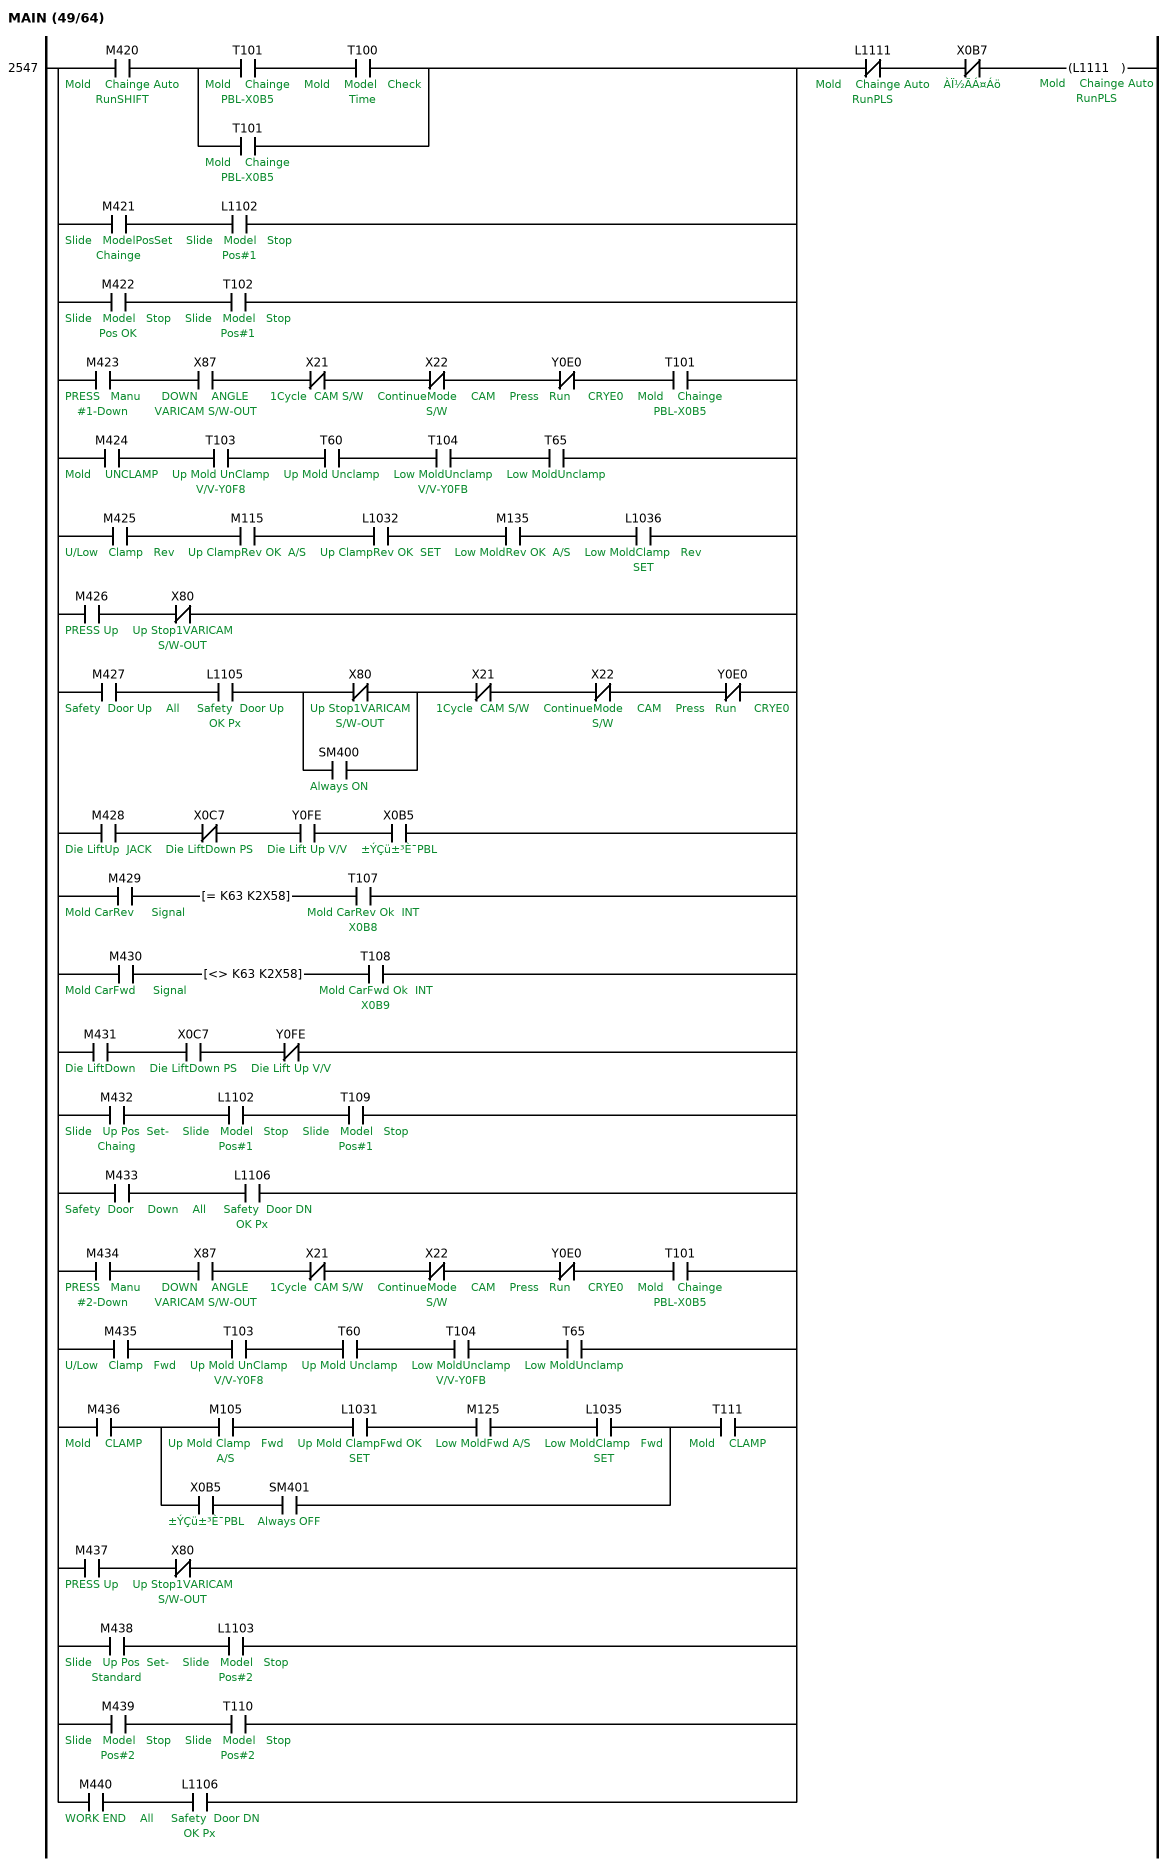
[picture p48: ladder of MAIN, rungs at steps 2547 to 2547]
2547  LD      M420  ; Mold    Chainge Auto RunSHIFT
      LD      T101  ; Mold    Chainge PBL-X0B5
      AND     T100  ; Mold    Model   Check   Time
      OR      T101  ; Mold    Chainge PBL-X0B5
      ANB
      LD      M421  ; Slide   ModelPosSet     Chainge
      AND     L1102  ; Slide   Model   Stop    Pos#1
      ORB
      LD      M422  ; Slide   Model   Stop    Pos OK
      AND     T102  ; Slide   Model   Stop    Pos#1
      ORB
      LD      M423  ; PRESS   Manu #1-Down
      AND     X87  ; DOWN    ANGLE   VARICAM S/W-OUT
      ANI     X21  ; 1Cycle  CAM S/W
      ANI     X22  ; ContinueMode    CAM S/W
      ANI     Y0E0  ; Press   Run     CRYE0
      AND     T101  ; Mold    Chainge PBL-X0B5
      ORB
      LD      M424  ; Mold    UNCLAMP
      AND     T103  ; Up Mold UnClamp V/V-Y0F8
      AND     T60  ; Up Mold Unclamp
      AND     T104  ; Low MoldUnclamp V/V-Y0FB
      AND     T65  ; Low MoldUnclamp
      ORB
      LD      M425  ; U/Low   Clamp   Rev
      AND     M115  ; Up ClampRev OK  A/S
      AND     L1032  ; Up ClampRev OK  SET
      AND     M135  ; Low MoldRev OK  A/S
      AND     L1036  ; Low MoldClamp   Rev SET
      ORB
      LD      M426  ; PRESS Up
      ANI     X80  ; Up Stop1VARICAM S/W-OUT
      ORB
      LD      M427  ; Safety  Door Up
      AND     L1105  ; All     Safety  Door Up OK Px
      LDI     X80  ; Up Stop1VARICAM S/W-OUT
      OR      SM400  ; Always ON
      ANB
      ANI     X21  ; 1Cycle  CAM S/W
      ANI     X22  ; ContinueMode    CAM S/W
      ANI     Y0E0  ; Press   Run     CRYE0
      ORB
      LD      M428  ; Die LiftUp  JACK
      ANI     X0C7  ; Die LiftDown PS
      AND     Y0FE  ; Die Lift Up V/V
      AND     X0B5  ; ±ÝÇü±³È¯PBL
      ORB
      LD      M429  ; Mold CarRev     Signal
      AND=    K63 K2X58
      AND     T107  ; Mold CarRev Ok  INT X0B8
      ORB
      LD      M430  ; Mold CarFwd     Signal
      AND<>   K63 K2X58
      AND     T108  ; Mold CarFwd Ok  INT X0B9
      ORB
      LD      M431  ; Die LiftDown
      AND     X0C7  ; Die LiftDown PS
      ANI     Y0FE  ; Die Lift Up V/V
      ORB
      LD      M432  ; Slide   Up Pos  Set-    Chaing
      AND     L1102  ; Slide   Model   Stop    Pos#1
      AND     T109  ; Slide   Model   Stop    Pos#1
      ORB
      LD      M433  ; Safety  Door    Down
      AND     L1106  ; All     Safety  Door DN OK Px
      ORB
      LD      M434  ; PRESS   Manu #2-Down
      AND     X87  ; DOWN    ANGLE   VARICAM S/W-OUT
      ANI     X21  ; 1Cycle  CAM S/W
      ANI     X22  ; ContinueMode    CAM S/W
      ANI     Y0E0  ; Press   Run     CRYE0
      AND     T101  ; Mold    Chainge PBL-X0B5
      ORB
      LD      M435  ; U/Low   Clamp   Fwd
      AND     T103  ; Up Mold UnClamp V/V-Y0F8
      AND     T60  ; Up Mold Unclamp
      AND     T104  ; Low MoldUnclamp V/V-Y0FB
      AND     T65  ; Low MoldUnclamp
      ORB
      LD      M436  ; Mold    CLAMP
      LD      M105  ; Up Mold Clamp   Fwd A/S
      AND     L1031  ; Up Mold ClampFwd OK  SET
      AND     M125  ; Low MoldFwd A/S
      AND     L1035  ; Low MoldClamp   Fwd SET
      LD      X0B5  ; ±ÝÇü±³È¯PBL
      AND     SM401  ; Always OFF
      ORB
      ANB
      AND     T111  ; Mold    CLAMP
      ORB
      LD      M437  ; PRESS Up
      ANI     X80  ; Up Stop1VARICAM S/W-OUT
      ORB
      LD      M438  ; Slide   Up Pos  Set-    Standard
      AND     L1103  ; Slide   Model   Stop    Pos#2
      ORB
      LD      M439  ; Slide   Model   Stop    Pos#2
      AND     T110  ; Slide   Model   Stop    Pos#2
      ORB
      LD      M440  ; WORK END
      AND     L1106  ; All     Safety  Door DN OK Px
      ORB
      ANI     L1111  ; Mold    Chainge Auto RunPLS
      ANI     X0B7  ; ÀÏ½ÃÁ¤Áö
      OUT     L1111  ; Mold    Chainge Auto RunPLS
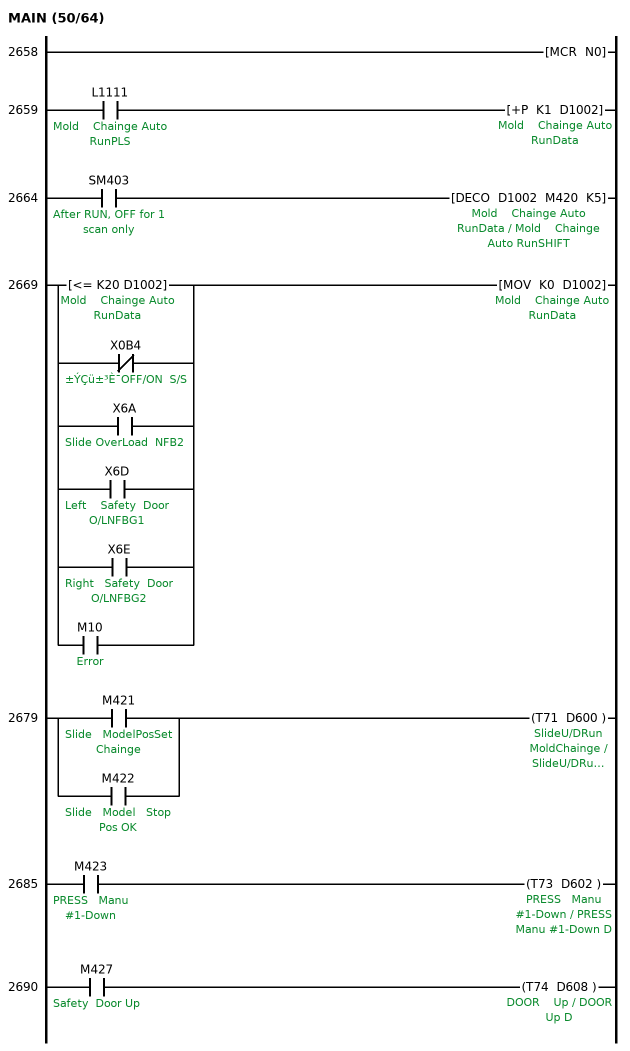
2658  MCR     N0
2659  LD      L1111  ; Mold    Chainge Auto RunPLS
      +P      K1 D1002  ; Mold    Chainge Auto RunData
2664  LD      SM403  ; After RUN, OFF for 1 scan only
      DECO    D1002 M420 K5
2669  LD<=    K20 D1002  ; Mold    Chainge Auto RunData
      ORI     X0B4  ; ±ÝÇü±³È¯OFF/ON  S/S
      OR      X6A  ; Slide OverLoad  NFB2
      OR      X6D  ; Left    Safety  Door O/LNFBG1
      OR      X6E  ; Right   Safety  Door O/LNFBG2
      OR      M10  ; Error
      MOV     K0 D1002
2679  LD      M421  ; Slide   ModelPosSet     Chainge
      OR      M422  ; Slide   Model   Stop    Pos OK
      OUT     T71 D600  ; SlideU/DRun MoldChainge / SlideU/DRun MoldChainge
2685  LD      M423  ; PRESS   Manu #1-Down
      OUT     T73 D602  ; PRESS   Manu #1-Down / PRESS   Manu #1-Down D
2690  LD      M427  ; Safety  Door Up
      OUT     T74 D608  ; DOOR    Up / DOOR    Up D
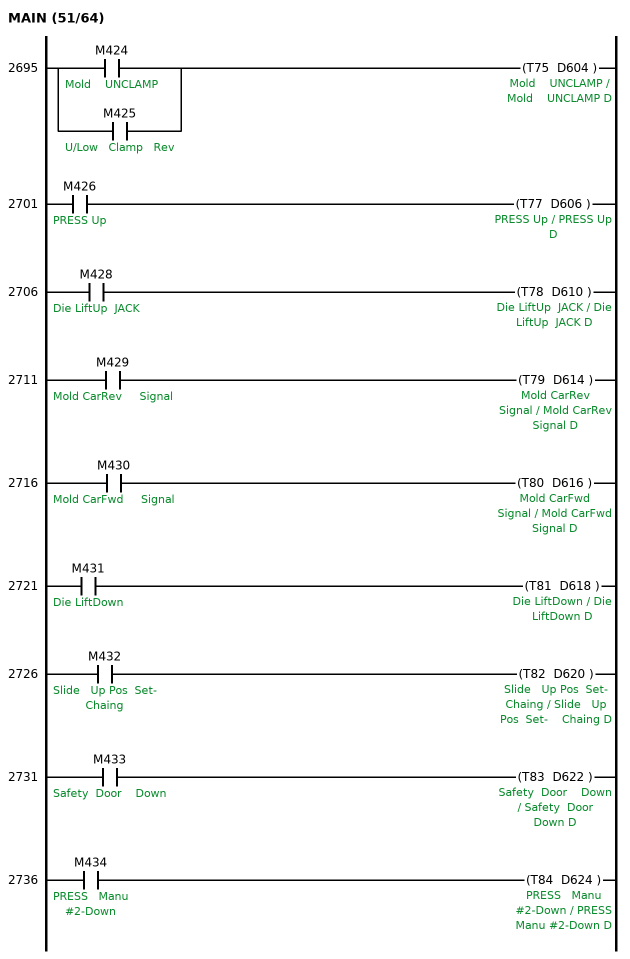
2695  LD      M424  ; Mold    UNCLAMP
      OR      M425  ; U/Low   Clamp   Rev
      OUT     T75 D604  ; Mold    UNCLAMP / Mold    UNCLAMP D
2701  LD      M426  ; PRESS Up
      OUT     T77 D606  ; PRESS Up / PRESS Up D
2706  LD      M428  ; Die LiftUp  JACK
      OUT     T78 D610  ; Die LiftUp  JACK / Die LiftUp  JACK D
2711  LD      M429  ; Mold CarRev     Signal
      OUT     T79 D614  ; Mold CarRev     Signal / Mold CarRev     Signal D
2716  LD      M430  ; Mold CarFwd     Signal
      OUT     T80 D616  ; Mold CarFwd     Signal / Mold CarFwd     Signal D
2721  LD      M431  ; Die LiftDown
      OUT     T81 D618  ; Die LiftDown / Die LiftDown D
2726  LD      M432  ; Slide   Up Pos  Set-    Chaing
      OUT     T82 D620  ; Slide   Up Pos  Set-    Chaing / Slide   Up Pos  Set-    Chaing D
2731  LD      M433  ; Safety  Door    Down
      OUT     T83 D622  ; Safety  Door    Down / Safety  Door    Down D
2736  LD      M434  ; PRESS   Manu #2-Down
      OUT     T84 D624  ; PRESS   Manu #2-Down / PRESS   Manu #2-Down D
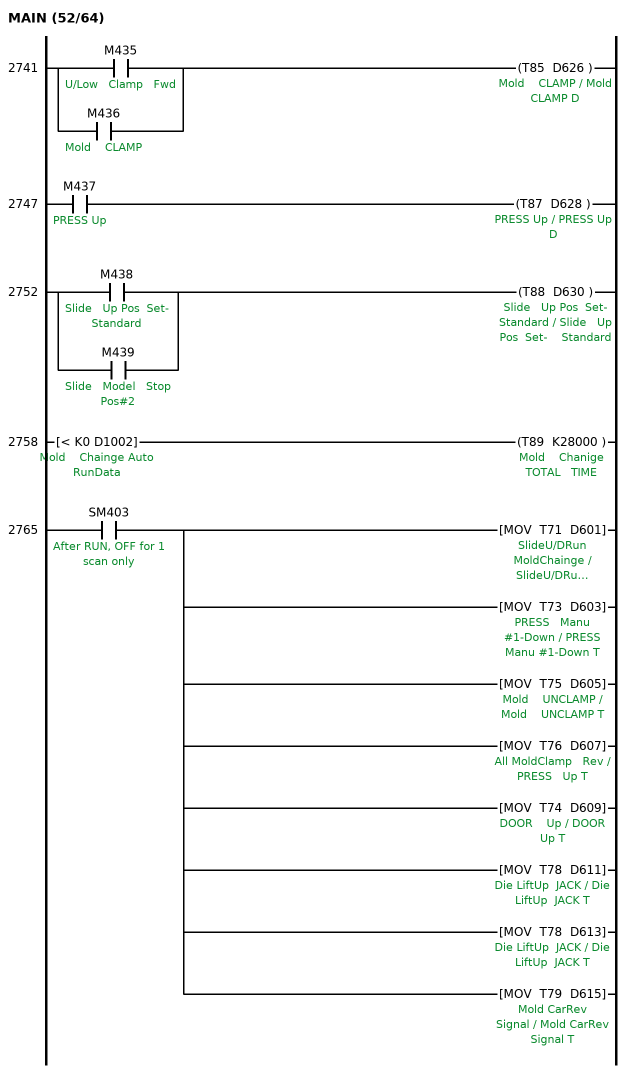
2741  LD      M435  ; U/Low   Clamp   Fwd
      OR      M436  ; Mold    CLAMP
      OUT     T85 D626  ; Mold    CLAMP / Mold    CLAMP D
2747  LD      M437  ; PRESS Up
      OUT     T87 D628  ; PRESS Up / PRESS Up D
2752  LD      M438  ; Slide   Up Pos  Set-    Standard
      OR      M439  ; Slide   Model   Stop    Pos#2
      OUT     T88 D630  ; Slide   Up Pos  Set-    Standard / Slide   Up Pos  Set-    Standard
2758  LD<     K0 D1002  ; Mold    Chainge Auto RunData
      OUT     T89 K28000  ; Mold    Chanige TOTAL   TIME
2765  LD      SM403  ; After RUN, OFF for 1 scan only
      MOV     T71 D601  ; SlideU/DRun MoldChainge T
      MOV     T73 D603  ; PRESS   Manu #1-Down T
      MOV     T75 D605  ; Mold    UNCLAMP T
      MOV     T76 D607  ; All MoldClamp   Rev / PRESS   Up T
      MOV     T74 D609  ; DOOR    Up T
      MOV     T78 D611  ; Die LiftUp  JACK T
      MOV     T78 D613  ; Die LiftUp  JACK T
      MOV     T79 D615  ; Mold CarRev     Signal T
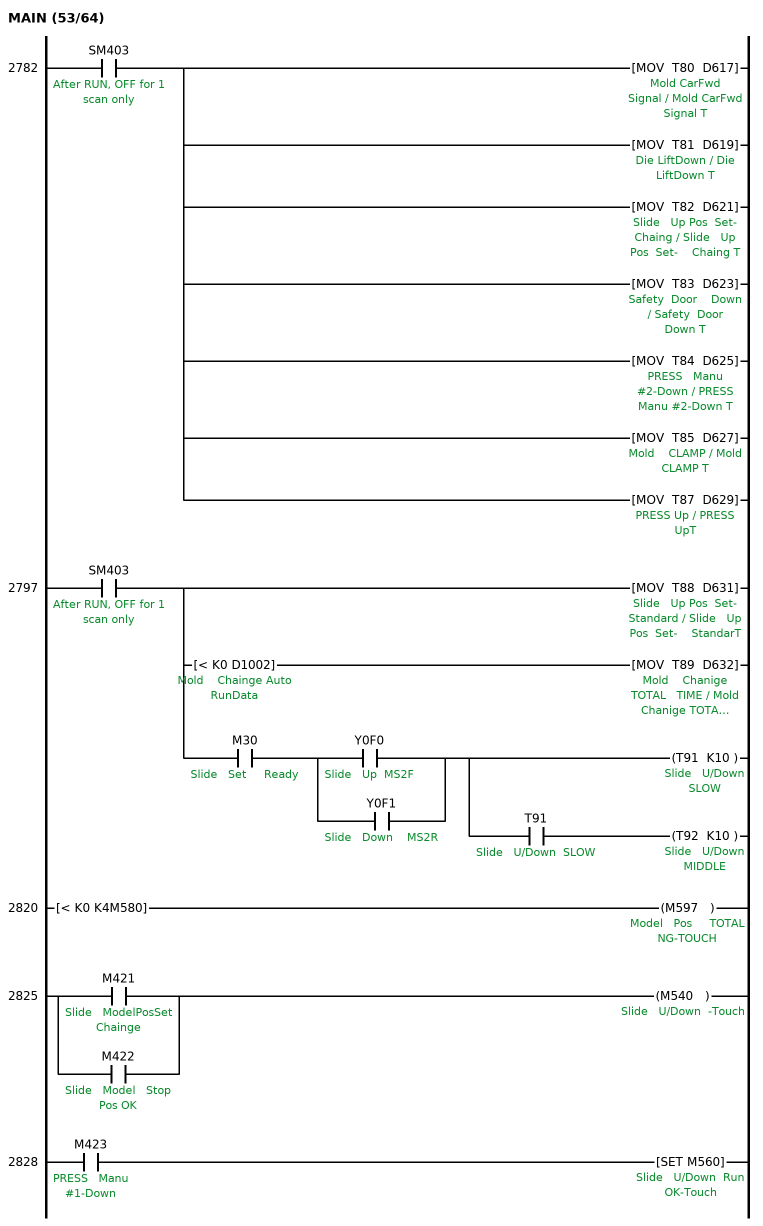
2782  LD      SM403  ; After RUN, OFF for 1 scan only
      MOV     T80 D617  ; Mold CarFwd     Signal T
      MOV     T81 D619  ; Die LiftDown T
      MOV     T82 D621  ; Slide   Up Pos  Set-    Chaing T
      MOV     T83 D623  ; Safety  Door    Down T
      MOV     T84 D625  ; PRESS   Manu #2-Down T
      MOV     T85 D627  ; Mold    CLAMP T
      MOV     T87 D629  ; PRESS UpT
2797  LD      SM403  ; After RUN, OFF for 1 scan only
      MOV     T88 D631  ; Slide   Up Pos  Set-    StandarT
      MPS
      AND<    K0 D1002  ; Mold    Chainge Auto RunData
      MOV     T89 D632  ; Mold    Chanige TOTAL   TIME
      MPP
      AND     M30  ; Slide   Set     Ready
      LD      Y0F0  ; Slide   Up  MS2F
      OR      Y0F1  ; Slide   Down    MS2R
      ANB
      OUT     T91 K10  ; Slide   U/Down  SLOW
      AND     T91  ; Slide   U/Down  SLOW
      OUT     T92 K10  ; Slide   U/Down  MIDDLE
2820  LD<     K0 K4M580  ; Slide   U/Down  Run   NG-Touch
      OUT     M597  ; Model   Pos     TOTAL   NG-TOUCH
2825  LD      M421  ; Slide   ModelPosSet     Chainge
      OR      M422  ; Slide   Model   Stop    Pos OK
      OUT     M540  ; Slide   U/Down  -Touch
2828  LD      M423  ; PRESS   Manu #1-Down
      SET     M560  ; Slide   U/Down  Run   OK-Touch
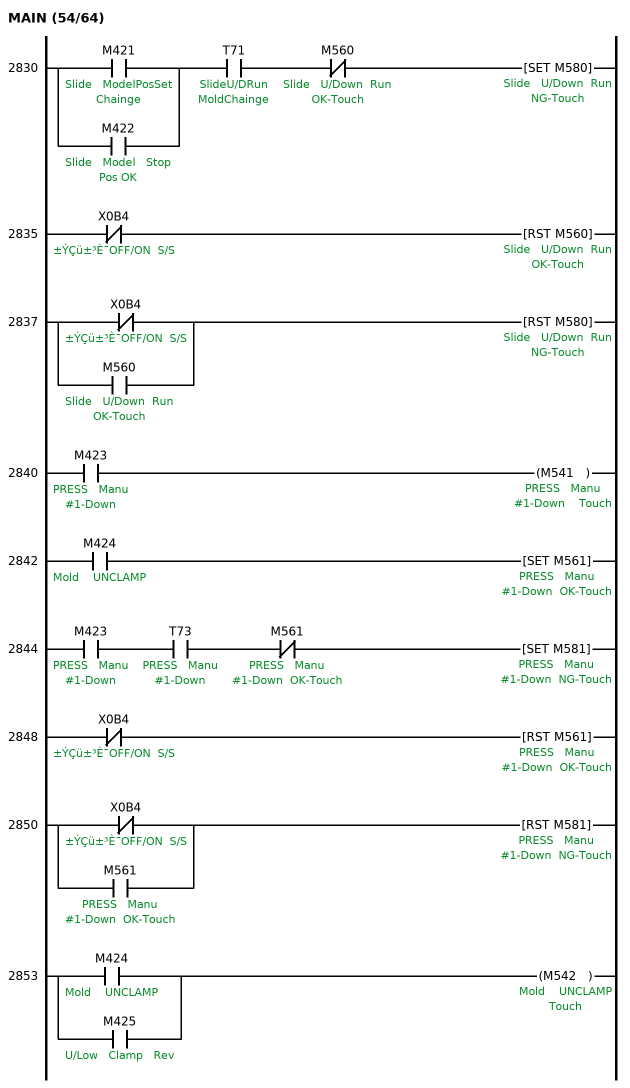
2830  LD      M421  ; Slide   ModelPosSet     Chainge
      OR      M422  ; Slide   Model   Stop    Pos OK
      AND     T71  ; SlideU/DRun MoldChainge
      ANI     M560  ; Slide   U/Down  Run   OK-Touch
      SET     M580  ; Slide   U/Down  Run   NG-Touch
2835  LDI     X0B4  ; ±ÝÇü±³È¯OFF/ON  S/S
      RST     M560  ; Slide   U/Down  Run   OK-Touch
2837  LDI     X0B4  ; ±ÝÇü±³È¯OFF/ON  S/S
      OR      M560  ; Slide   U/Down  Run   OK-Touch
      RST     M580  ; Slide   U/Down  Run   NG-Touch
2840  LD      M423  ; PRESS   Manu #1-Down
      OUT     M541  ; PRESS   Manu #1-Down    Touch
2842  LD      M424  ; Mold    UNCLAMP
      SET     M561  ; PRESS   Manu #1-Down  OK-Touch
2844  LD      M423  ; PRESS   Manu #1-Down
      AND     T73  ; PRESS   Manu #1-Down
      ANI     M561  ; PRESS   Manu #1-Down  OK-Touch
      SET     M581  ; PRESS   Manu #1-Down  NG-Touch
2848  LDI     X0B4  ; ±ÝÇü±³È¯OFF/ON  S/S
      RST     M561  ; PRESS   Manu #1-Down  OK-Touch
2850  LDI     X0B4  ; ±ÝÇü±³È¯OFF/ON  S/S
      OR      M561  ; PRESS   Manu #1-Down  OK-Touch
      RST     M581  ; PRESS   Manu #1-Down  NG-Touch
2853  LD      M424  ; Mold    UNCLAMP
      OR      M425  ; U/Low   Clamp   Rev
      OUT     M542  ; Mold    UNCLAMP Touch
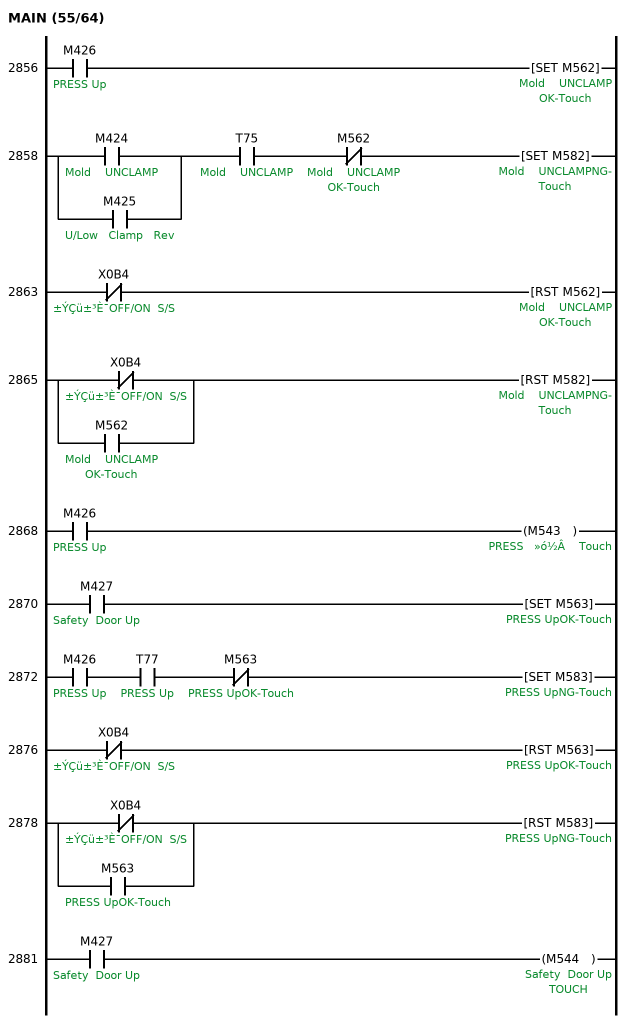
2856  LD      M426  ; PRESS Up
      SET     M562  ; Mold    UNCLAMP OK-Touch
2858  LD      M424  ; Mold    UNCLAMP
      OR      M425  ; U/Low   Clamp   Rev
      AND     T75  ; Mold    UNCLAMP
      ANI     M562  ; Mold    UNCLAMP OK-Touch
      SET     M582  ; Mold    UNCLAMPNG-Touch
2863  LDI     X0B4  ; ±ÝÇü±³È¯OFF/ON  S/S
      RST     M562  ; Mold    UNCLAMP OK-Touch
2865  LDI     X0B4  ; ±ÝÇü±³È¯OFF/ON  S/S
      OR      M562  ; Mold    UNCLAMP OK-Touch
      RST     M582  ; Mold    UNCLAMPNG-Touch
2868  LD      M426  ; PRESS Up
      OUT     M543  ; PRESS   »ó½Â    Touch
2870  LD      M427  ; Safety  Door Up
      SET     M563  ; PRESS UpOK-Touch
2872  LD      M426  ; PRESS Up
      AND     T77  ; PRESS Up
      ANI     M563  ; PRESS UpOK-Touch
      SET     M583  ; PRESS UpNG-Touch
2876  LDI     X0B4  ; ±ÝÇü±³È¯OFF/ON  S/S
      RST     M563  ; PRESS UpOK-Touch
2878  LDI     X0B4  ; ±ÝÇü±³È¯OFF/ON  S/S
      OR      M563  ; PRESS UpOK-Touch
      RST     M583  ; PRESS UpNG-Touch
2881  LD      M427  ; Safety  Door Up
      OUT     M544  ; Safety  Door Up TOUCH
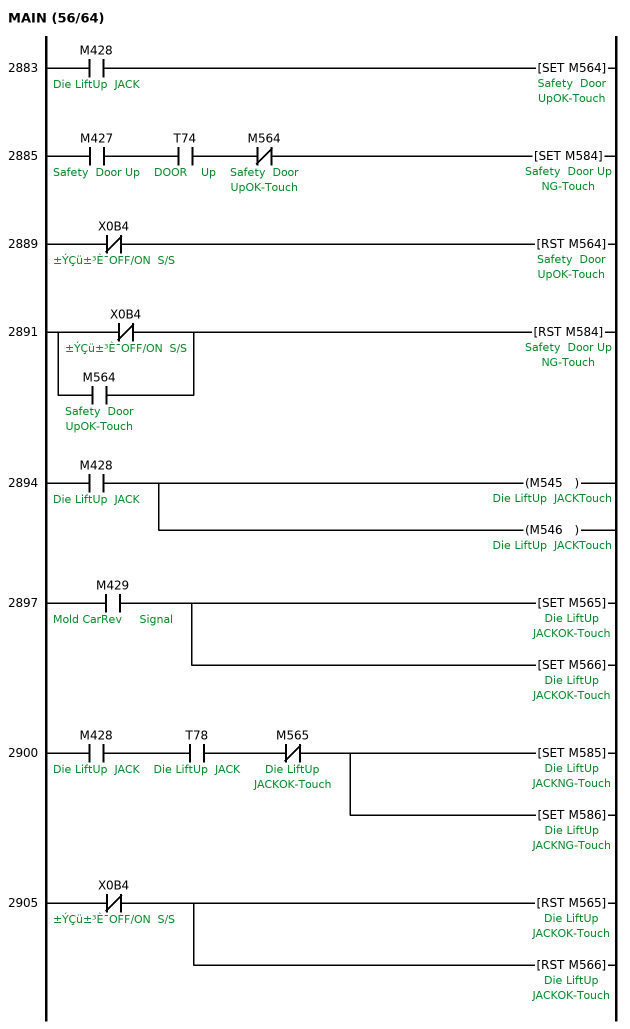
2883  LD      M428  ; Die LiftUp  JACK
      SET     M564  ; Safety  Door UpOK-Touch
2885  LD      M427  ; Safety  Door Up
      AND     T74  ; DOOR    Up
      ANI     M564  ; Safety  Door UpOK-Touch
      SET     M584  ; Safety  Door Up NG-Touch
2889  LDI     X0B4  ; ±ÝÇü±³È¯OFF/ON  S/S
      RST     M564  ; Safety  Door UpOK-Touch
2891  LDI     X0B4  ; ±ÝÇü±³È¯OFF/ON  S/S
      OR      M564  ; Safety  Door UpOK-Touch
      RST     M584  ; Safety  Door Up NG-Touch
2894  LD      M428  ; Die LiftUp  JACK
      OUT     M545  ; Die LiftUp  JACKTouch
      OUT     M546  ; Die LiftUp  JACKTouch
2897  LD      M429  ; Mold CarRev     Signal
      SET     M565  ; Die LiftUp  JACKOK-Touch
      SET     M566  ; Die LiftUp  JACKOK-Touch
2900  LD      M428  ; Die LiftUp  JACK
      AND     T78  ; Die LiftUp  JACK
      ANI     M565  ; Die LiftUp  JACKOK-Touch
      SET     M585  ; Die LiftUp  JACKNG-Touch
      SET     M586  ; Die LiftUp  JACKNG-Touch
2905  LDI     X0B4  ; ±ÝÇü±³È¯OFF/ON  S/S
      RST     M565  ; Die LiftUp  JACKOK-Touch
      RST     M566  ; Die LiftUp  JACKOK-Touch
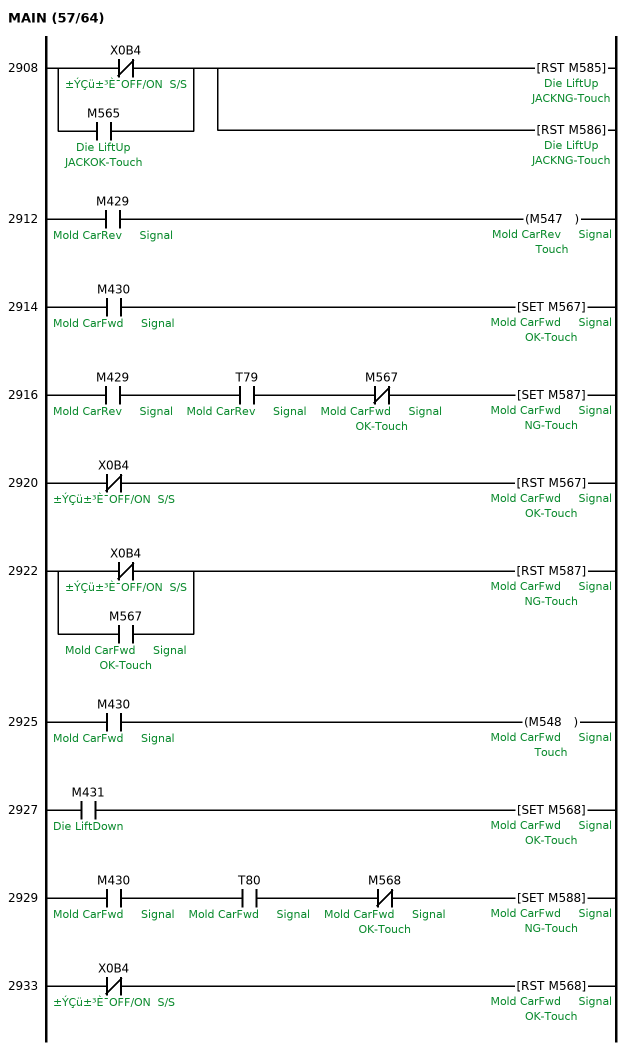
2908  LDI     X0B4  ; ±ÝÇü±³È¯OFF/ON  S/S
      OR      M565  ; Die LiftUp  JACKOK-Touch
      RST     M585  ; Die LiftUp  JACKNG-Touch
      RST     M586  ; Die LiftUp  JACKNG-Touch
2912  LD      M429  ; Mold CarRev     Signal
      OUT     M547  ; Mold CarRev     Signal  Touch
2914  LD      M430  ; Mold CarFwd     Signal
      SET     M567  ; Mold CarFwd     Signal  OK-Touch
2916  LD      M429  ; Mold CarRev     Signal
      AND     T79  ; Mold CarRev     Signal
      ANI     M567  ; Mold CarFwd     Signal  OK-Touch
      SET     M587  ; Mold CarFwd     Signal  NG-Touch
2920  LDI     X0B4  ; ±ÝÇü±³È¯OFF/ON  S/S
      RST     M567  ; Mold CarFwd     Signal  OK-Touch
2922  LDI     X0B4  ; ±ÝÇü±³È¯OFF/ON  S/S
      OR      M567  ; Mold CarFwd     Signal  OK-Touch
      RST     M587  ; Mold CarFwd     Signal  NG-Touch
2925  LD      M430  ; Mold CarFwd     Signal
      OUT     M548  ; Mold CarFwd     Signal  Touch
2927  LD      M431  ; Die LiftDown
      SET     M568  ; Mold CarFwd     Signal  OK-Touch
2929  LD      M430  ; Mold CarFwd     Signal
      AND     T80  ; Mold CarFwd     Signal
      ANI     M568  ; Mold CarFwd     Signal  OK-Touch
      SET     M588  ; Mold CarFwd     Signal  NG-Touch
2933  LDI     X0B4  ; ±ÝÇü±³È¯OFF/ON  S/S
      RST     M568  ; Mold CarFwd     Signal  OK-Touch
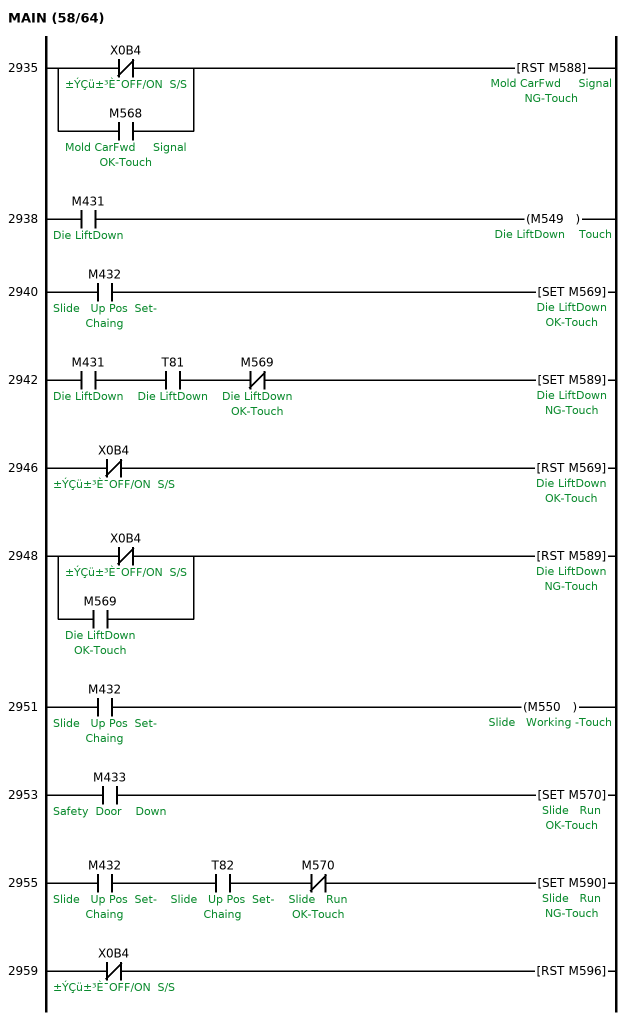
2935  LDI     X0B4  ; ±ÝÇü±³È¯OFF/ON  S/S
      OR      M568  ; Mold CarFwd     Signal  OK-Touch
      RST     M588  ; Mold CarFwd     Signal  NG-Touch
2938  LD      M431  ; Die LiftDown
      OUT     M549  ; Die LiftDown    Touch
2940  LD      M432  ; Slide   Up Pos  Set-    Chaing
      SET     M569  ; Die LiftDown    OK-Touch
2942  LD      M431  ; Die LiftDown
      AND     T81  ; Die LiftDown
      ANI     M569  ; Die LiftDown    OK-Touch
      SET     M589  ; Die LiftDown    NG-Touch
2946  LDI     X0B4  ; ±ÝÇü±³È¯OFF/ON  S/S
      RST     M569  ; Die LiftDown    OK-Touch
2948  LDI     X0B4  ; ±ÝÇü±³È¯OFF/ON  S/S
      OR      M569  ; Die LiftDown    OK-Touch
      RST     M589  ; Die LiftDown    NG-Touch
2951  LD      M432  ; Slide   Up Pos  Set-    Chaing
      OUT     M550  ; Slide   Working -Touch
2953  LD      M433  ; Safety  Door    Down
      SET     M570  ; Slide   Run     OK-Touch
2955  LD      M432  ; Slide   Up Pos  Set-    Chaing
      AND     T82  ; Slide   Up Pos  Set-    Chaing
      ANI     M570  ; Slide   Run     OK-Touch
      SET     M590  ; Slide   Run     NG-Touch
2959  LDI     X0B4  ; ±ÝÇü±³È¯OFF/ON  S/S
      RST     M596
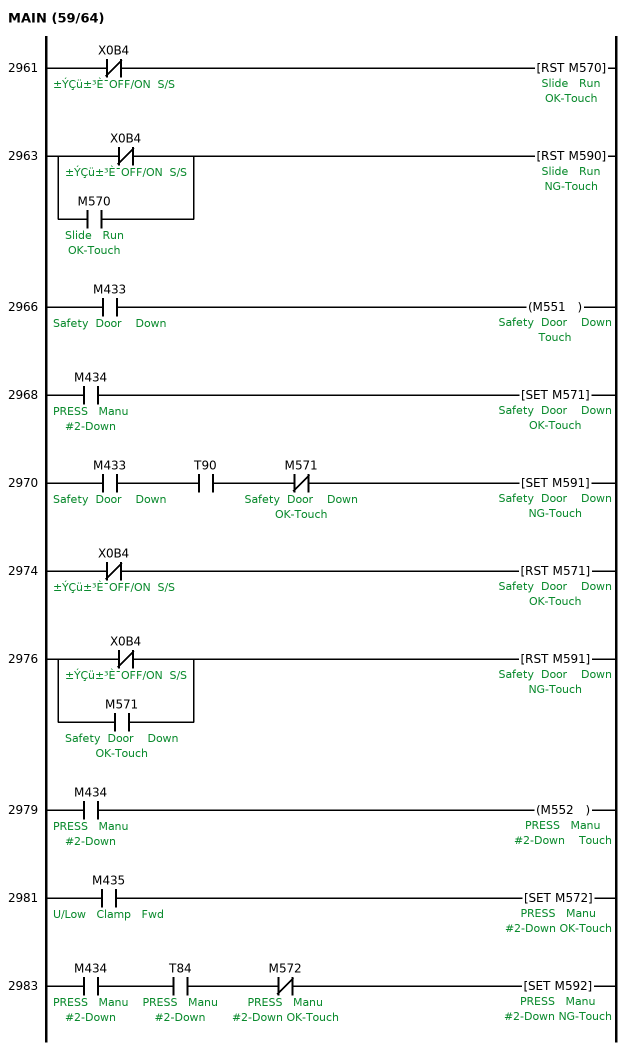
2961  LDI     X0B4  ; ±ÝÇü±³È¯OFF/ON  S/S
      RST     M570  ; Slide   Run     OK-Touch
2963  LDI     X0B4  ; ±ÝÇü±³È¯OFF/ON  S/S
      OR      M570  ; Slide   Run     OK-Touch
      RST     M590  ; Slide   Run     NG-Touch
2966  LD      M433  ; Safety  Door    Down
      OUT     M551  ; Safety  Door    Down    Touch
2968  LD      M434  ; PRESS   Manu #2-Down
      SET     M571  ; Safety  Door    Down    OK-Touch
2970  LD      M433  ; Safety  Door    Down
      AND     T90
      ANI     M571  ; Safety  Door    Down    OK-Touch
      SET     M591  ; Safety  Door    Down    NG-Touch
2974  LDI     X0B4  ; ±ÝÇü±³È¯OFF/ON  S/S
      RST     M571  ; Safety  Door    Down    OK-Touch
2976  LDI     X0B4  ; ±ÝÇü±³È¯OFF/ON  S/S
      OR      M571  ; Safety  Door    Down    OK-Touch
      RST     M591  ; Safety  Door    Down    NG-Touch
2979  LD      M434  ; PRESS   Manu #2-Down
      OUT     M552  ; PRESS   Manu #2-Down    Touch
2981  LD      M435  ; U/Low   Clamp   Fwd
      SET     M572  ; PRESS   Manu #2-Down OK-Touch
2983  LD      M434  ; PRESS   Manu #2-Down
      AND     T84  ; PRESS   Manu #2-Down
      ANI     M572  ; PRESS   Manu #2-Down OK-Touch
      SET     M592  ; PRESS   Manu #2-Down NG-Touch
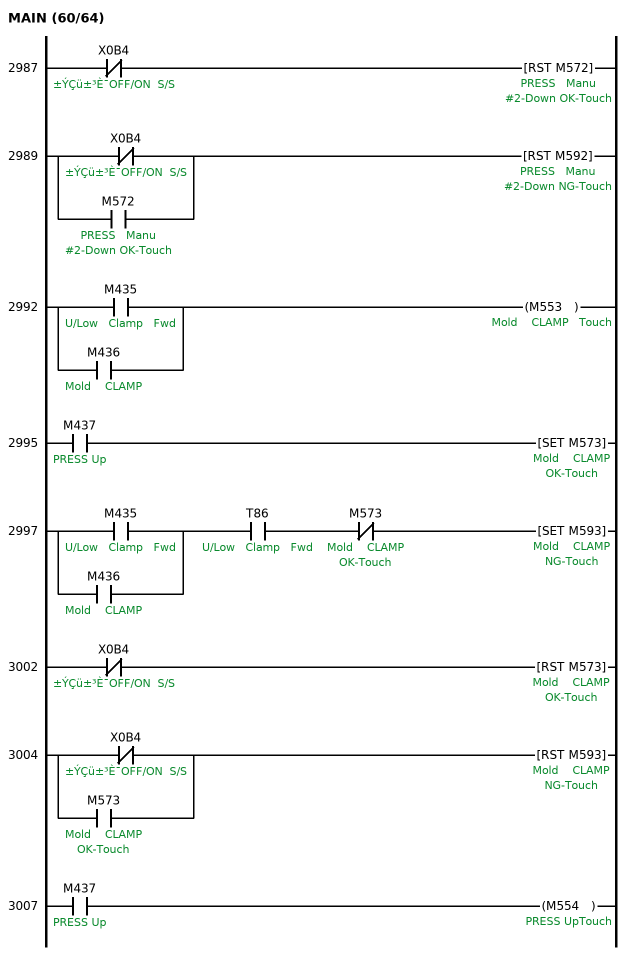
2987  LDI     X0B4  ; ±ÝÇü±³È¯OFF/ON  S/S
      RST     M572  ; PRESS   Manu #2-Down OK-Touch
2989  LDI     X0B4  ; ±ÝÇü±³È¯OFF/ON  S/S
      OR      M572  ; PRESS   Manu #2-Down OK-Touch
      RST     M592  ; PRESS   Manu #2-Down NG-Touch
2992  LD      M435  ; U/Low   Clamp   Fwd
      OR      M436  ; Mold    CLAMP
      OUT     M553  ; Mold    CLAMP   Touch
2995  LD      M437  ; PRESS Up
      SET     M573  ; Mold    CLAMP   OK-Touch
2997  LD      M435  ; U/Low   Clamp   Fwd
      OR      M436  ; Mold    CLAMP
      AND     T86  ; U/Low   Clamp   Fwd
      ANI     M573  ; Mold    CLAMP   OK-Touch
      SET     M593  ; Mold    CLAMP   NG-Touch
3002  LDI     X0B4  ; ±ÝÇü±³È¯OFF/ON  S/S
      RST     M573  ; Mold    CLAMP   OK-Touch
3004  LDI     X0B4  ; ±ÝÇü±³È¯OFF/ON  S/S
      OR      M573  ; Mold    CLAMP   OK-Touch
      RST     M593  ; Mold    CLAMP   NG-Touch
3007  LD      M437  ; PRESS Up
      OUT     M554  ; PRESS UpTouch
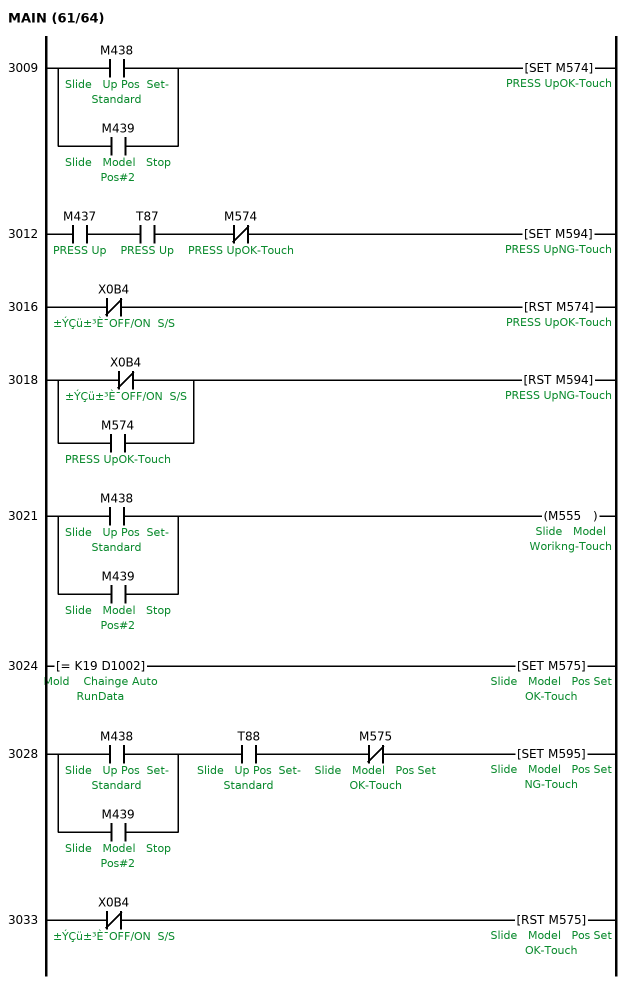
3009  LD      M438  ; Slide   Up Pos  Set-    Standard
      OR      M439  ; Slide   Model   Stop    Pos#2
      SET     M574  ; PRESS UpOK-Touch
3012  LD      M437  ; PRESS Up
      AND     T87  ; PRESS Up
      ANI     M574  ; PRESS UpOK-Touch
      SET     M594  ; PRESS UpNG-Touch
3016  LDI     X0B4  ; ±ÝÇü±³È¯OFF/ON  S/S
      RST     M574  ; PRESS UpOK-Touch
3018  LDI     X0B4  ; ±ÝÇü±³È¯OFF/ON  S/S
      OR      M574  ; PRESS UpOK-Touch
      RST     M594  ; PRESS UpNG-Touch
3021  LD      M438  ; Slide   Up Pos  Set-    Standard
      OR      M439  ; Slide   Model   Stop    Pos#2
      OUT     M555  ; Slide   Model   Worikng-Touch
3024  LD=     K19 D1002  ; Mold    Chainge Auto RunData
      SET     M575  ; Slide   Model   Pos Set OK-Touch
3028  LD      M438  ; Slide   Up Pos  Set-    Standard
      OR      M439  ; Slide   Model   Stop    Pos#2
      AND     T88  ; Slide   Up Pos  Set-    Standard
      ANI     M575  ; Slide   Model   Pos Set OK-Touch
      SET     M595  ; Slide   Model   Pos Set NG-Touch
3033  LDI     X0B4  ; ±ÝÇü±³È¯OFF/ON  S/S
      RST     M575  ; Slide   Model   Pos Set OK-Touch
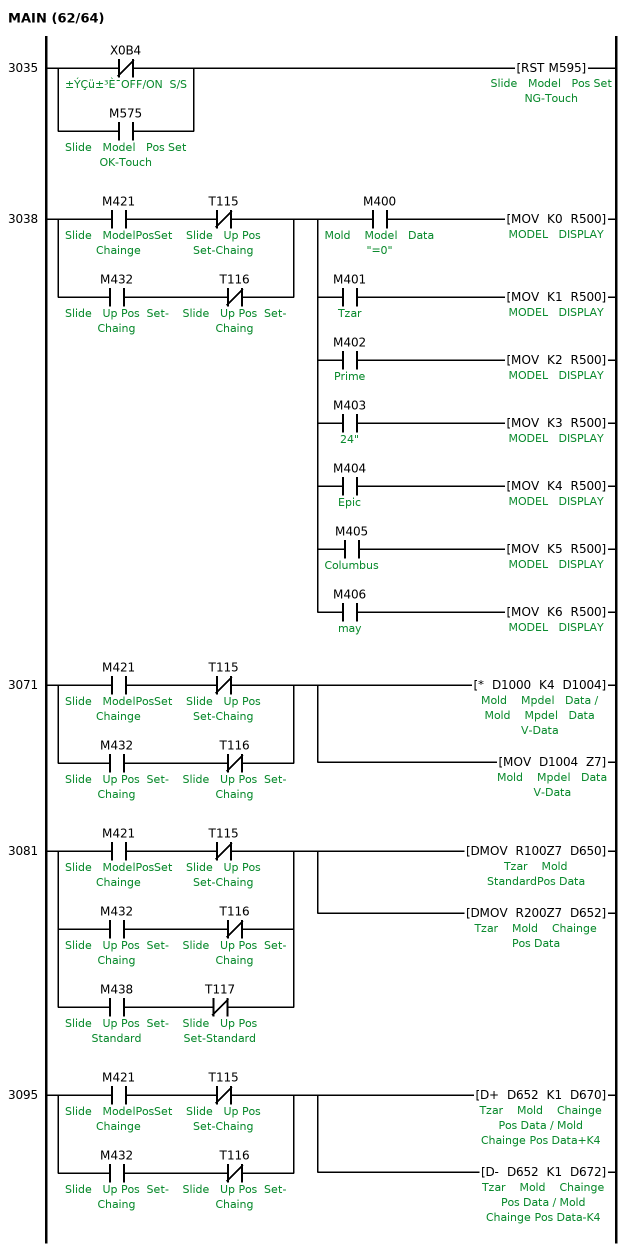
3035  LDI     X0B4  ; ±ÝÇü±³È¯OFF/ON  S/S
      OR      M575  ; Slide   Model   Pos Set OK-Touch
      RST     M595  ; Slide   Model   Pos Set NG-Touch
3038  LD      M421  ; Slide   ModelPosSet     Chainge
      ANI     T115  ; Slide   Up Pos  Set-Chaing
      LD      M432  ; Slide   Up Pos  Set-    Chaing
      ANI     T116  ; Slide   Up Pos  Set-    Chaing
      ORB
      MPS
      AND     M400  ; Mold    Model   Data    "=0"
      MOV     K0 R500  ; MODEL   DISPLAY
      MRD
      AND     M401  ; Tzar
      MOV     K1 R500
      MRD
      AND     M402  ; Prime
      MOV     K2 R500
      MRD
      AND     M403  ; 24"
      MOV     K3 R500
      MRD
      AND     M404  ; Epic
      MOV     K4 R500
      MRD
      AND     M405  ; Columbus
      MOV     K5 R500
      MPP
      AND     M406  ; may
      MOV     K6 R500
3071  LD      M421  ; Slide   ModelPosSet     Chainge
      ANI     T115  ; Slide   Up Pos  Set-Chaing
      LD      M432  ; Slide   Up Pos  Set-    Chaing
      ANI     T116  ; Slide   Up Pos  Set-    Chaing
      ORB
      *       D1000 K4 D1004  ; Mold    Mpdel   Data    V-Data
      MOV     D1004 Z7
3081  LD      M421  ; Slide   ModelPosSet     Chainge
      ANI     T115  ; Slide   Up Pos  Set-Chaing
      LD      M432  ; Slide   Up Pos  Set-    Chaing
      ANI     T116  ; Slide   Up Pos  Set-    Chaing
      ORB
      LD      M438  ; Slide   Up Pos  Set-    Standard
      ANI     T117  ; Slide   Up Pos  Set-Standard
      ORB
      DMOV    R100Z7 D650  ; Tzar    Mold    StandardPos Data
      DMOV    R200Z7 D652  ; Tzar    Mold    Chainge Pos Data
3095  LD      M421  ; Slide   ModelPosSet     Chainge
      ANI     T115  ; Slide   Up Pos  Set-Chaing
      LD      M432  ; Slide   Up Pos  Set-    Chaing
      ANI     T116  ; Slide   Up Pos  Set-    Chaing
      ORB
      D+      D652 K1 D670
      D-      D652 K1 D672
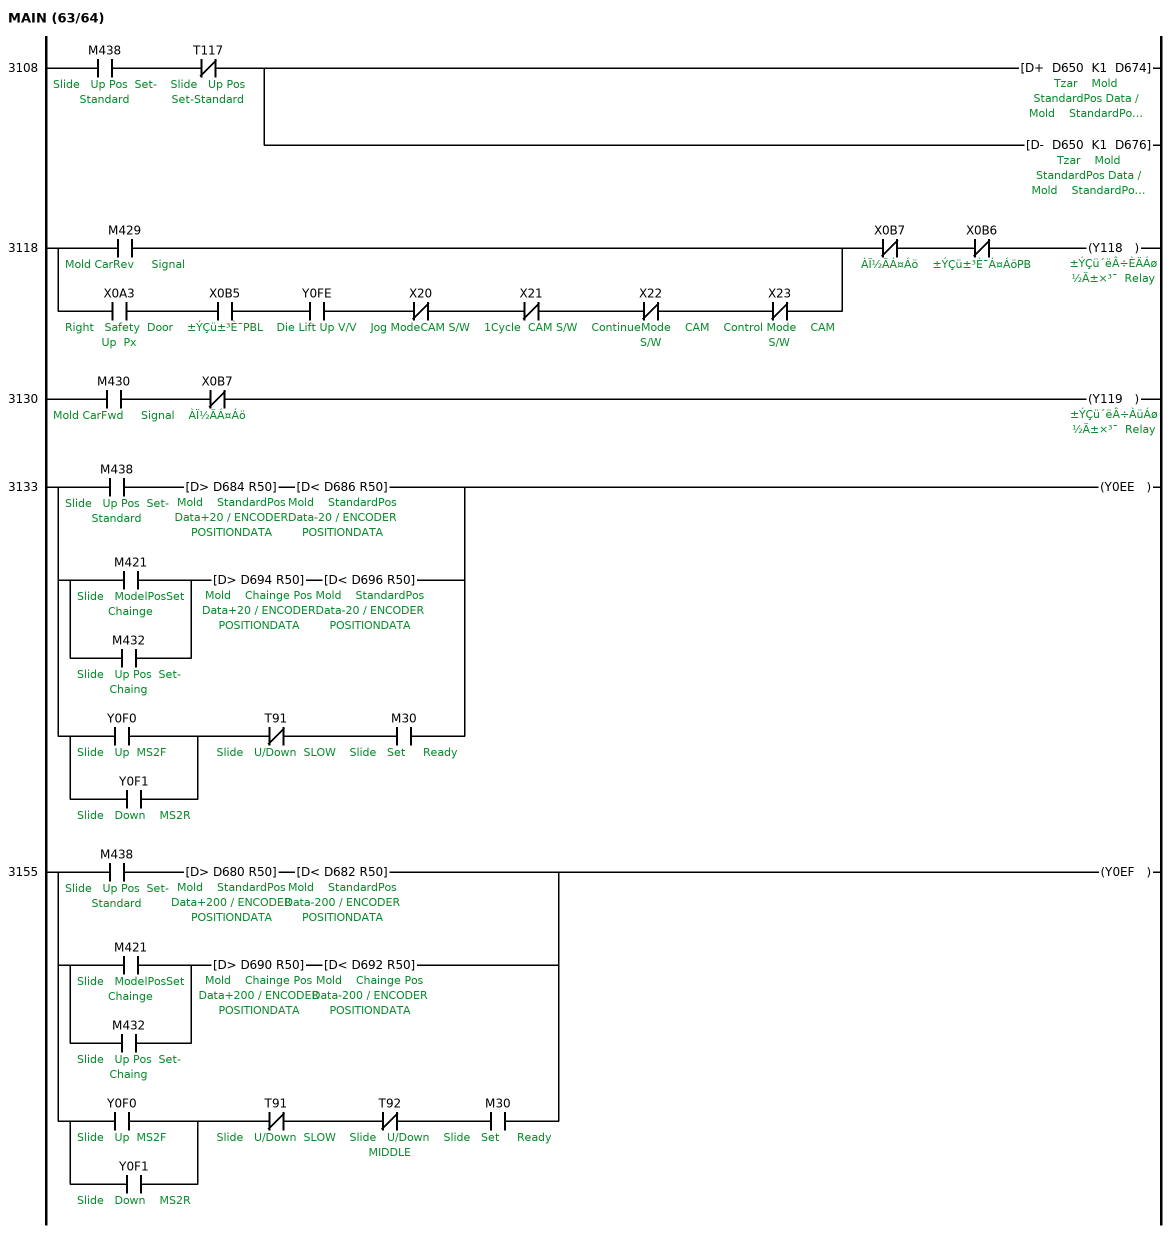
3108  LD      M438  ; Slide   Up Pos  Set-    Standard
      ANI     T117  ; Slide   Up Pos  Set-Standard
      D+      D650 K1 D674
      D-      D650 K1 D676
3118  LD      M429  ; Mold CarRev     Signal
      LD      X0A3  ; Right   Safety  Door Up  Px
      AND     X0B5  ; ±ÝÇü±³È¯PBL
      AND     Y0FE  ; Die Lift Up V/V
      ANI     X20  ; Jog ModeCAM S/W
      ANI     X21  ; 1Cycle  CAM S/W
      ANI     X22  ; ContinueMode    CAM S/W
      ANI     X23  ; Control Mode    CAM S/W
      ORB
      ANI     X0B7  ; ÀÏ½ÃÁ¤Áö
      ANI     X0B6  ; ±ÝÇü±³È¯Á¤ÁöPB
      OUT     Y118  ; ±ÝÇü´ëÂ÷ÈÄÁø    ½Ã±×³¯  Relay
3130  LD      M430  ; Mold CarFwd     Signal
      ANI     X0B7  ; ÀÏ½ÃÁ¤Áö
      OUT     Y119  ; ±ÝÇü´ëÂ÷ÀüÁø    ½Ã±×³¯  Relay
3133  LD      M438  ; Slide   Up Pos  Set-    Standard
      ANDD>   D684 R50  ; Mold    StandardPos Data+20 / ENCODER POSITIONDATA
      ANDD<   D686 R50  ; Mold    StandardPos Data-20 / ENCODER POSITIONDATA
      LD      M421  ; Slide   ModelPosSet     Chainge
      OR      M432  ; Slide   Up Pos  Set-    Chaing
      ANDD>   D694 R50  ; Mold    Chainge Pos Data+20 / ENCODER POSITIONDATA
      ANDD<   D696 R50  ; Mold    StandardPos Data-20 / ENCODER POSITIONDATA
      ORB
      LD      Y0F0  ; Slide   Up  MS2F
      OR      Y0F1  ; Slide   Down    MS2R
      ANI     T91  ; Slide   U/Down  SLOW
      AND     M30  ; Slide   Set     Ready
      ORB
      OUT     Y0EE
3155  LD      M438  ; Slide   Up Pos  Set-    Standard
      ANDD>   D680 R50  ; Mold    StandardPos Data+200 / ENCODER POSITIONDATA
      ANDD<   D682 R50  ; Mold    StandardPos Data-200 / ENCODER POSITIONDATA
      LD      M421  ; Slide   ModelPosSet     Chainge
      OR      M432  ; Slide   Up Pos  Set-    Chaing
      ANDD>   D690 R50  ; Mold    Chainge Pos Data+200 / ENCODER POSITIONDATA
      ANDD<   D692 R50  ; Mold    Chainge Pos Data-200 / ENCODER POSITIONDATA
      ORB
      LD      Y0F0  ; Slide   Up  MS2F
      OR      Y0F1  ; Slide   Down    MS2R
      ANI     T91  ; Slide   U/Down  SLOW
      ANI     T92  ; Slide   U/Down  MIDDLE
      AND     M30  ; Slide   Set     Ready
      ORB
      OUT     Y0EF
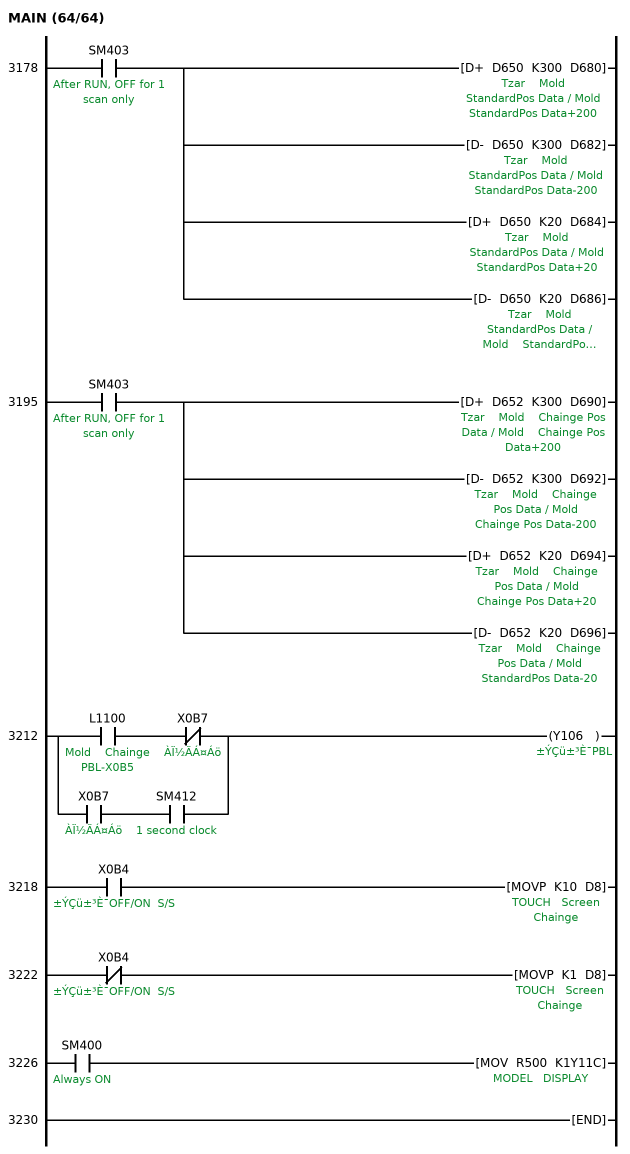
3178  LD      SM403  ; After RUN, OFF for 1 scan only
      D+      D650 K300 D680
      D-      D650 K300 D682
      D+      D650 K20 D684
      D-      D650 K20 D686
3195  LD      SM403  ; After RUN, OFF for 1 scan only
      D+      D652 K300 D690
      D-      D652 K300 D692
      D+      D652 K20 D694
      D-      D652 K20 D696
3212  LD      L1100  ; Mold    Chainge PBL-X0B5
      ANI     X0B7  ; ÀÏ½ÃÁ¤Áö
      LD      X0B7  ; ÀÏ½ÃÁ¤Áö
      AND     SM412  ; 1 second clock
      ORB
      OUT     Y106  ; ±ÝÇü±³È¯PBL
3218  LD      X0B4  ; ±ÝÇü±³È¯OFF/ON  S/S
      MOVP    K10 D8  ; TOUCH   Screen  Chainge
3222  LDI     X0B4  ; ±ÝÇü±³È¯OFF/ON  S/S
      MOVP    K1 D8
3226  LD      SM400  ; Always ON
      MOV     R500 K1Y11C
3230  END
END_PROGRAM
